INTERFACE I_Directory

// Deletes files in the directory that were created before the provided date.
METHOD DeleteFilesCreatedBefore : BOOL
VAR_INPUT
	path				: Tc2_System.T_MaxString;	// Path to where the deletion should be performed
	fileNameContains	: Tc2_System.T_MaxString;	// Some characters that the file name should containt
	netId				: Tc2_System.T_AmsNetID;	// NetId where the search should occurr
	thresholdDate		: DT;	// If created before this date, the file will be deleted.
END_VAR

VAR_OUTPUT
	error			: BOOL;
	errorInfo		: ZigaLibs_Core.ST_AdsError;	
	deletedFiles	: ARRAY[0..100] OF Tc2_System.T_MaxString;	// A list of deleted items, as T_MaxString (file names).
END_VAR
END_METHOD

// Looks if the provided directory exists on the disk.
// Returns TRUE when done
// Result can be found in the output directoryExists.
METHOD Exists : BOOL
VAR_INPUT
	directory	: Tc2_System.T_MaxString;	// Path to the directory that will be searched.
	netId		: Tc2_System.T_AmsNetID;	// NetId where to search.
END_VAR

VAR_OUTPUT
	directoryExists		: BOOL;	// TRUE if it exists, else FALSE. Only valid after method returns TRUE.
END_VAR
END_METHOD

(* Looks in the directory `path` and iterates the content. 
 When method returns TRUE, the collection of items is found in the result I_Collection.*)
METHOD ListAll : BOOL
VAR_INPUT
	path	: Tc2_System.T_MaxString;	// Path to the directory that will be searched.
	netId	: Tc2_System.T_AmsNetID;	// NetId where to search.
END_VAR

VAR_IN_OUT
	items	: ARRAY[*] OF Tc2_Utilities.ST_FindFileEntry;	// Collection of found files in the provided location	
END_VAR

VAR_OUTPUT
	error		: BOOL;	// Will be true if an error occurs while executing the file query
	errorInfo	: ZigaLibs_Core.ST_AdsError;	// Error information will be provided here
END_VAR
END_METHOD

(* Looks in the directory `path` and iterates the content. 
 When method returns TRUE, the collection of files is found in the result I_Collection.*)
METHOD ListFiles : BOOL
VAR_INPUT
	path	: Tc2_System.T_MaxString;	// Path to the directory that will be searched.
	netId	: Tc2_System.T_AmsNetID;	// NetId where to search.
END_VAR

VAR_IN_OUT
	files	: ARRAY[*] OF Tc2_System.T_MaxString;	// Collection of found files in the provided location.
END_VAR

VAR_OUTPUT
	error		: BOOL;	// Will be true if an error occurs while executing the file query
	errorInfo	: ZigaLibs_Core.ST_AdsError;	// Error information will be provided here
END_VAR
END_METHOD

END_INTERFACE

(* stored: Version 1.1.0.1, ProductVersion 3.1.4024.15
   Itf I_Directory: Id {cb7661a0-6c20-02b0-24ea-9f5626ca673d}
   Method DeleteFilesCreatedBefore: Id {98d738a9-600c-0c8f-3444-91bf4e5c4a7f}
   Method Exists: Id {1827d2ba-6c87-0271-0d65-2147c8b7d1dc}
   Method ListAll: Id {8957fa17-2e01-0184-32c2-bd2509e71d55}
   Method ListFiles: Id {c1dba3ed-539c-00f4-3c7d-1830c5959103} *)
